{attribute 'GeneratedUsingTerminal: IL2302-B110-0017'}
{attribute addProperty BoxType "IL2302-B110-0017"}
{attribute addProperty Id "Term_24KL_D4CFBC220Term_395_Ix1000KL_8EF4D3E90"}
{attribute addProperty CRC "3784109104"}
{attribute addProperty Size "0"}
TYPE A_0024_IL2302_B110_0017_E18CEC30 EXTENDS IL2302_13409EDF :
STRUCT
	{attribute addProperty Name "Term_24"}
	Term_24 : KL_D4CFBC22;
	{attribute addProperty Name "Term_395_Ix1000"}
	Term_395_Ix1000 : KL_8EF4D3E9;
END_STRUCT
END_TYPE

(* stored: Version 1.2.0.0, ProductVersion 3.1.4024.9
   DUT A_0024_IL2302_B110_0017_E18CEC30: Id {3e9fe7ed-dfee-44bc-ae95-7e89d3ac613d} *)
